{attribute 'OPC.UA.DA.StructuredType' := '1'}
TYPE ST_MotomanCtrl_out :
STRUCT	
	Error	: UINT;
END_STRUCT
END_TYPE

(* stored: Version 1.1.0.1, ProductVersion 3.1.4024.9
   DUT ST_MotomanCtrl_out: Id {7f187a9d-c84c-4354-b0b2-765942f5f27d} *)
